Staubli VAL3: iLidClosed.pgx

public program iLidClosed(num& nNum[] (dimensions=1))
begin
  nNum=dioGet(iLidClosed)
end
